FUNCTION_BLOCK MyCalculatorClass
VAR
END_VAR

METHOD Divide : INT
VAR_INPUT
	x : INT;
	y : INT;
END_VAR
IF y <> 0 THEN
	Divide := x/y;
ELSE
	Divide := -1;
END_IF
END_METHOD

END_FUNCTION_BLOCK

(* stored: Version 1.1.0.1, ProductVersion 3.1.4024.12
   POU MyCalculatorClass: Id {e4bd4153-2e3b-4816-9317-28aa7cb3f8b8}, SpecialFunc None
   Method Divide: Id {bc7e5332-51ef-40d3-92e0-2f2f2eba9f96} *)
